Staubli VAL3: onF7Event.pgx

program onF7Event()
  local string l_sMessage
  local num l_nType
begin
  // look if the bButton is enable
  if bButton[6]
    //
    //  Delete the selected process
    //
    call processList:getDefaultType(l_nType)
    call processList:delete(nIndex,l_nType)
    logMsg("[KERNEL] INTERFACE:Delete the program: "+sEvent+" at the index: "+toString("",nIndex))
    if nIndex==0 and cycleStatus:bCycle
      call OnEvent:endCycle()
      call language:message(l_sMessage,3)
      popUpMsg(l_sMessage)
    endIf
  endIf
end
